// TIA Portal project "Loop_Traffic_Light" (V18)

(* hardware
DEVICE "S7-1500/ET200MP station_1"  S7-1500 station
   slot 0: "导轨_0"  Rack  6ES7 590-1***0-0AA0
   slot 1: "PLC_1"  CPU 1516-3 PN/DP  6ES7 516-3AN01-0AB0  V2.6
      slot 3: "CPU 显示_1"  6ES7591-1BA00-0AA0
      slot 32768: "PROFINET 接口_1"  X1
      slot 33024: "PROFINET 接口_2"  X2
      slot 33280: "DP 接口_1"  X3
   slot 2: "DI 32x24VDC HF_1"  DI 32x24VDC HF  6ES7 521-1BL00-0AB0  V2.1
   slot 3: "DQ 32x24VDC/0.5A HF_1"  DQ 32x24VDC/0.5A HF  6ES7 522-1BL01-0AB0  V1.1
   slot 4: "AI 8xU/I/RTD/TC ST_1"  AI 8xU/I/RTD/TC ST  6ES7 531-7KF00-0AB0  V2.2
   slot 5: "AQ 4xU/I ST_1"  AQ 4xU/I ST  6ES7 532-5HD00-0AB0  V2.2
DEVICE "HMI_1"  TP700 Comfort
   slot 0: "HMI_1"  TP700 Comfort  6AV2 124-0GC01-0AX0  15.1.0.0
   slot 1: "HMI_RT_1"  TP700 Comfort  6AV2 124-0GC01-0AX0  15.1.0.0
   slot 5: "HMI_1.IE_CP_1"  PROFINET Interface  15.0.1.0
      slot 1: "PROFINET Interface_1"  PROFINET Interface
         slot 1: "Port_1"  Port
         slot 2: "Port_2"  Port
   slot 7: "HMI_1.MPI/DP_CP_1"  MPI/DP Interface  15.0.1.0
*)

// ===== PLC "PLC_1"  CPU 1516-3 PN/DP =====

VAR_GLOBAL   // PLC tag table "默认变量表"
   "System_Byte" AT %MB1 : Byte;
   "FirstScan" AT %M1.0 : Bool;
   "DiagStatusUpdate" AT %M1.1 : Bool;
   "AlwaysTRUE" AT %M1.2 : Bool;
   "AlwaysFALSE" AT %M1.3 : Bool;
   "Clock_Byte" AT %MB0 : Byte;
   "Clock_10Hz" AT %M0.0 : Bool;
   "Clock_5Hz" AT %M0.1 : Bool;
   "Clock_2.5Hz" AT %M0.2 : Bool;
   "Clock_2Hz" AT %M0.3 : Bool;
   "Clock_1.25Hz" AT %M0.4 : Bool;
   "Clock_1Hz" AT %M0.5 : Bool;
   "Clock_0.625Hz" AT %M0.6 : Bool;
   "Clock_0.5Hz" AT %M0.7 : Bool;
   "启动按钮" AT %I1.0 : Bool;   // 蓝色按钮
   "急停按钮" AT %I1.5 : Bool;   // 红色按钮
   "黄灯" AT %Q1.1 : Bool;
   "绿灯" AT %Q1.2 : Bool;
   "红灯" AT %Q1.3 : Bool;
   "启动标志" AT %M10.0 : Bool;
   "时钟" AT %M20.0 : Bool;
   "T5_R" AT %M10.3 : Bool;
   "灯循环" AT %M10.1 : Bool;
   "Tag_1" AT %Q1.0 : Bool;
   "Tag_3" AT %T2 : Timer;
   "T1_R" AT %M10.4 : Bool;
   "T2_R" AT %M10.5 : Bool;
   "循环次数" AT %MW100 : Word;
   "Tag_2" AT %M30.0 : Bool;
   "Tag_4" AT %M20.1 : Bool;
   "Tag_5" AT %M20.2 : Bool;
END_VAR

DATA_BLOCK "块_1_DB"   // DB6
{ S7_Optimized_Access := 'TRUE' }
VERSION : 0.1
// stored: InstanceOfName 块_1
"块_1"
BEGIN
END_DATA_BLOCK

// folder: System blocks/Program resources

DATA_BLOCK "T1"   // DB1
{ S7_Optimized_Access := 'TRUE' }
AUTHOR : Simatic
FAMILY : IEC
NAME : IEC_TMR
VERSION : 1.0
// stored: InstanceOfName IEC_TIMER
"IEC_TIMER"
BEGIN
END_DATA_BLOCK

DATA_BLOCK "T2"   // DB2
{ S7_Optimized_Access := 'TRUE' }
AUTHOR : Simatic
FAMILY : IEC
NAME : IEC_TMR
VERSION : 1.0
// stored: InstanceOfName IEC_TIMER
"IEC_TIMER"
BEGIN
END_DATA_BLOCK

DATA_BLOCK "T3"   // DB3
{ S7_Optimized_Access := 'TRUE' }
AUTHOR : Simatic
FAMILY : IEC
NAME : IEC_TMR
VERSION : 1.0
// stored: InstanceOfName IEC_TIMER
"IEC_TIMER"
BEGIN
END_DATA_BLOCK

DATA_BLOCK "T4"   // DB4
{ S7_Optimized_Access := 'TRUE' }
AUTHOR : Simatic
FAMILY : IEC
NAME : IEC_TMR
VERSION : 1.0
// stored: InstanceOfName IEC_TIMER
"IEC_TIMER"
BEGIN
END_DATA_BLOCK

DATA_BLOCK "T5"   // DB5
{ S7_Optimized_Access := 'TRUE' }
AUTHOR : Simatic
FAMILY : IEC
NAME : IEC_TMR
VERSION : 1.0
// stored: InstanceOfName IEC_TIMER
"IEC_TIMER"
BEGIN
END_DATA_BLOCK

DATA_BLOCK "T6"   // DB7
{ S7_Optimized_Access := 'TRUE' }
AUTHOR : Simatic
FAMILY : IEC
NAME : IEC_TMR
VERSION : 1.0
// stored: InstanceOfName IEC_TIMER
"IEC_TIMER"
BEGIN
END_DATA_BLOCK

// folder: (top level)

FUNCTION_BLOCK "块_1"   // FB1, LAD
{ S7_Optimized_Access := 'TRUE' }
VERSION : 0.1
   VAR_TEMP   // added for the SCL form of the ladder/FBD networks
      _w1 : Bool;
   END_VAR
BEGIN

REGION Network 1
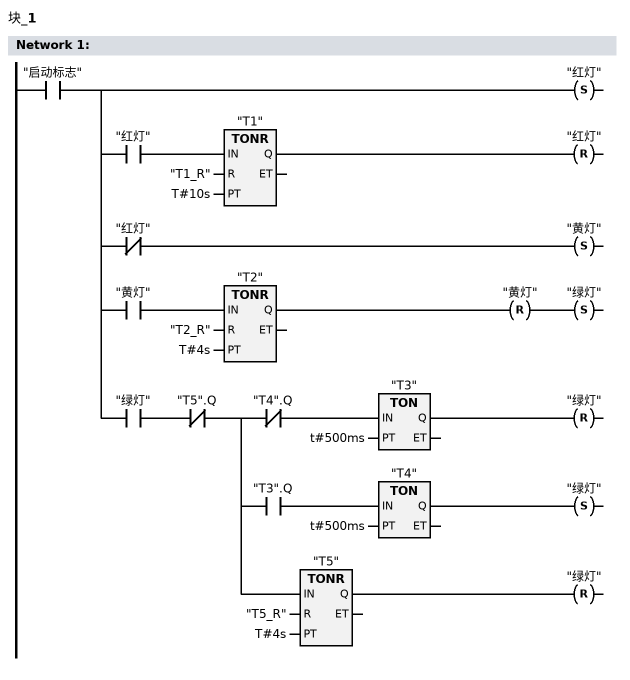
   IF "启动标志" THEN "红灯" := TRUE; END_IF;
   "T1".TONR(IN := "启动标志" AND "红灯", R := "T1_R", PT := T#10s);
   IF "T1".Q THEN "红灯" := FALSE; END_IF;
   IF "启动标志" AND NOT "红灯" THEN "黄灯" := TRUE; END_IF;
   "T2".TONR(IN := "启动标志" AND "黄灯", R := "T2_R", PT := T#4s);
   IF "T2".Q THEN
       "黄灯" := FALSE;
       "绿灯" := TRUE;
   END_IF;
   #_w1 := "启动标志" AND "绿灯" AND NOT "T5".Q;
   "T3".TON(IN := #_w1 AND NOT "T4".Q, PT := t#500ms);
   IF "T3".Q THEN "绿灯" := FALSE; END_IF;
   "T4".TON(IN := #_w1 AND "T3".Q, PT := t#500ms);
   IF "T4".Q THEN "绿灯" := TRUE; END_IF;
   "T5".TONR(IN := #_w1, R := "T5_R", PT := T#4s);
   IF "T5".Q THEN "绿灯" := FALSE; END_IF;
END_REGION
END_FUNCTION_BLOCK

ORGANIZATION_BLOCK "Main"   // OB1, LAD, ProgramCycle
TITLE = "Main Program Sweep (Cycle)"
{ S7_Optimized_Access := 'TRUE' }
VERSION : 0.1
   VAR_INPUT
      Initial_Call : Bool;   // Initial call of this OB
      Remanence : Bool;   // =True, if remanent data are available
   END_VAR
   VAR_TEMP   // added for the SCL form of the ladder/FBD networks
      _w1 : Bool;
   END_VAR
BEGIN

REGION Network 1: 启动_停止
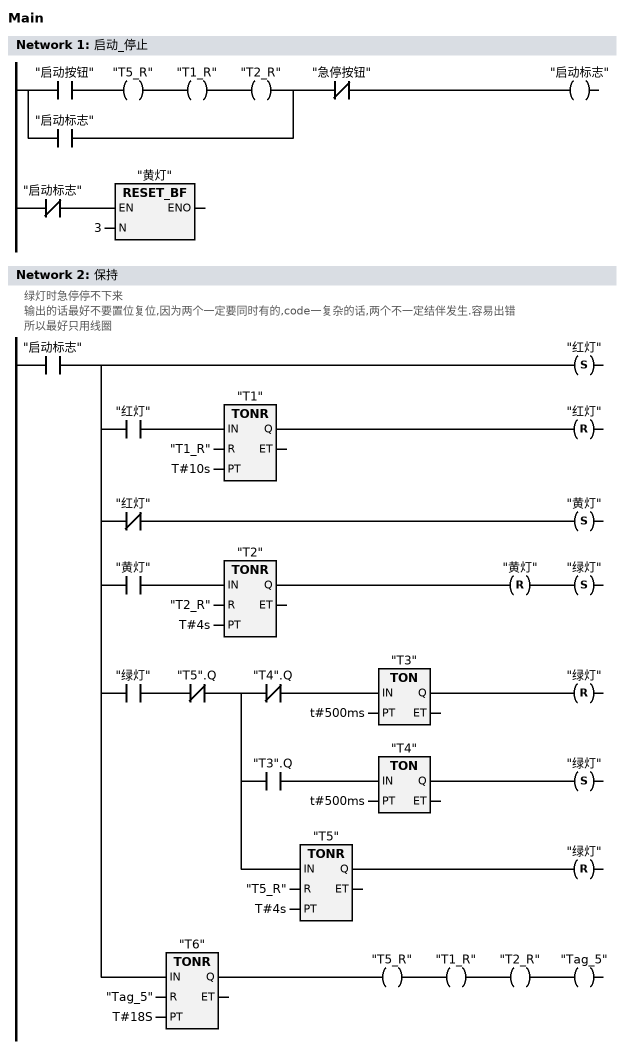
   // no SCL statement known for RBitfield: written as a call
   "T5_R" := "启动按钮";
   "T1_R" := "启动按钮";
   "T2_R" := "启动按钮";
   "启动标志" := ("启动按钮" OR "启动标志") AND NOT "急停按钮";
   IF NOT "启动标志" THEN RESET_BF(operand := "黄灯", n := 3); END_IF;
END_REGION

REGION Network 2: 保持
   // 绿灯时急停停不下来
   // 输出的话最好不要置位复位,因为两个一定要同时有的,code一复杂的话,两个不一定结伴发生.容易出错
   // 所以最好只用线圈
   IF "启动标志" THEN "红灯" := TRUE; END_IF;
   "T1".TONR(IN := "启动标志" AND "红灯", R := "T1_R", PT := T#10s);
   IF "T1".Q THEN "红灯" := FALSE; END_IF;
   IF "启动标志" AND NOT "红灯" THEN "黄灯" := TRUE; END_IF;
   "T2".TONR(IN := "启动标志" AND "黄灯", R := "T2_R", PT := T#4s);
   IF "T2".Q THEN
       "黄灯" := FALSE;
       "绿灯" := TRUE;
   END_IF;
   #_w1 := "启动标志" AND "绿灯" AND NOT "T5".Q;
   "T3".TON(IN := #_w1 AND NOT "T4".Q, PT := t#500ms);
   IF "T3".Q THEN "绿灯" := FALSE; END_IF;
   "T4".TON(IN := #_w1 AND "T3".Q, PT := t#500ms);
   IF "T4".Q THEN "绿灯" := TRUE; END_IF;
   "T5".TONR(IN := #_w1, R := "T5_R", PT := T#4s);
   IF "T5".Q THEN "绿灯" := FALSE; END_IF;
   "T6".TONR(IN := "启动标志", R := "Tag_5", PT := T#18S);
   "T5_R" := "T6".Q;
   "T1_R" := "T6".Q;
   "T2_R" := "T6".Q;
   "Tag_5" := "T6".Q;
END_REGION
END_ORGANIZATION_BLOCK

(* ===== HMI "HMI_RT_1" =====
system functions are stored by id; their names below are inferred from use
connection "HMI_连接_1": ETHERNET, S7_1500_OMS

HMI tags "默认变量表"
   "Tag_ScreenNumber" : UInt, internal
   "启动按钮" : Bool = PLC 启动按钮 AT %I1.0, 100 ms
   "急停按钮" : Bool = PLC 急停按钮 AT %I1.5, 100 ms
   "红灯" : Bool = PLC 红灯 AT %Q1.3, 100 ms
   "黄灯" : Bool = PLC 绿灯 AT %Q1.2, 100 ms
   "绿灯" : Bool = PLC 黄灯 AT %Q1.1, 100 ms

screen "根画面" 800x420, template "模板_1"
   on GenerateScreen: SetTag("Tag_ScreenNumber", 1)
   Button "按钮_1" at 200,75 size 96x32; TextOff '启动按钮'
      on Press: SetBit("启动按钮")
      on Release: ResetBit("启动按钮")
   Button "按钮_2" at 200,164 size 96x32; TextOff '急停按钮'
      on Press: SetBit("急停按钮")
      on Release: ResetBit("急停按钮")
   Circle "圆_1" at 423,103 size 48x48
      Appearance <- "红灯"
   Circle "圆_2" at 548,105 size 48x48
      Appearance <- "黄灯"
   Circle "圆_3" at 673,107 size 48x48
      Appearance <- "绿灯"
   TextField "文本域_1" at 423,69 size 39x20; Text '红灯'
   TextField "文本域_2" at 548,73 size 39x20; Text '黄灯'
   TextField "文本域_3" at 684,69 size 39x20; Text '绿灯'
   IOField "I/O 域_1" at 596,196 size 96x32; FormatPattern 9999999
   TextField "文本域_4" at 484,198 size 73x20; Text '循环次数'

Template "模板_1" 800x420
   Button "退出" at 720,360 size 78x58; TextOff '退出'; PictureOff "ExitRuntime_TP700_Comfort_TR"; PictureOn "ExitRuntime_TP700_Comfort_TR"
      on Release: StopRuntime(0)
   Button "Template_Button" at 640,360 size 78x58; TextOff 'Text'
   Button "Template_Button_1" at 560,360 size 78x58; TextOff 'Text'
   Button "Template_Button_2" at 480,360 size 78x58; TextOff 'Text'
   Button "Template_Button_3" at 400,360 size 78x58; TextOff 'Text'
   Button "Template_Button_4" at 321,360 size 78x58; TextOff 'Text'
   Button "Template_Button_5" at 241,360 size 78x58; TextOff 'Text'
   Button "Template_Button_6" at 161,360 size 78x58; TextOff 'Text'
   Button "报警" at 81,360 size 78x58; TextOff '报警'; PictureOff "AlarmDisplay_TP700_Comfort_TR"; PictureOn "AlarmDisplay_TP700_Comfort_TR"
      on Release: function_ef3f5d25("报警窗口_Unacknowledged", -1)
   Button "起始画面" at 1,360 size 78x58; TextOff '起始画面'; PictureOff "NavigateHome_TP700_Comfort_TR"; PictureOn "NavigateHome_TP700_Comfort_TR"
      on Release: ActivateScreen("根画面", 0)
*)